FUNCTION_BLOCK FB_AllocateRobotNeedlingMove EXTENDS FB_ActionBasic
VAR_INPUT
    xExecute      : BOOL;
    xAbort        : BOOL;
    TimeOut  : LREAL := 30; // Unit : s
	MovingInfo	: ST_AllocateRobotNeedlingMoveInfo;
END_VAR
VAR_OUTPUT
    xAborted : BOOL;
    iErrorID : INT;
    ErrorMsg : T_MaxString;
END_VAR
VAR
    StateBehavior   : CBML.ETrigATo;
    uiCyclicStep    : UINT := 0;
    uiIndexLoop     : UINT;
	Coordinate		:st_Coordinate;
	fbExecuteEdgeDetect :FB_EdgeDetect;
END_VAR

THIS^.IBehaviourModel := StateBehavior;
StateBehavior(xExecute := xExecute,
              xAbort := xAbort OR fbExecuteEdgeDetect.xFallingEdge,
              udiTimeOut := LREAL_TO_UDINT( TimeOut*1000000),
              xDone => xDone,
              xBusy => xBusy,
              xError => xError,			  
              xAborted => xAborted);			  

			  
//Make sure that C# turns off execute to shut down the service
fbExecuteEdgeDetect(xInput :=xExecute);

//Error Msg
iErrorID := StateBehavior._model.iErrorID;
ErrorMsg := M_GetErrorMsg(xErrorID := iErrorID);

METHOD CleanupAction
VAR_INPUT
    xAbortProposed : BOOL;
    iErrorIDProposed: INT;
END_VAR
VAR_OUTPUT
    xComplete : BOOL := TRUE;
    xAbort: BOOL := xAbortProposed;
 	iErrorID : INT := iErrorIDProposed;
END_VAR
uiCyclicStep := 0;
END_METHOD

METHOD CyclicAction
VAR_INPUT
    itfTimingController : CBML.ITimingController;
END_VAR
VAR_OUTPUT
    xComplete : BOOL := TRUE;
    iErrorID : INT := 0;
END_VAR
VAR_INST
	
END_VAR

VAR
		bAxesCheck 		: BOOL;
	
	
END_VAR
xComplete := FALSE;

	IF arAxisCtrl_gb[AxisNo.Allocate_X].Admin.Axis.Status.Error OR
		arAxisCtrl_gb[AxisNo.Allocate_Y].Admin.Axis.Status.Error THEN
		iErrorID :=3;
	END_IF

CASE uiCyclicStep OF
    0:
		
			uiCyclicStep:=100;
		
		
	100:
			arAxisCtrl_gb[AxisNo.Allocate_X].PosMode.Position:=Coordinate.X;
			arAxisCtrl_gb[AxisNo.Allocate_Y].PosMode.Position:=Coordinate.Y;	
		
			IF arAxisCtrl_gb[AxisNo.Allocate_X].Admin.Axis.Status.Moving OR
			   arAxisCtrl_gb[AxisNo.Allocate_Y].Admin.Axis.Status.Moving OR
			   arAxisStatus_gb[AxisNo.Allocate_X].Admin._OpModeAck=E_AXIS_MODE.ModePosAbs OR
			   arAxisStatus_gb[AxisNo.Allocate_y].Admin._OpModeAck=E_AXIS_MODE.ModePosAbs THEN
			   uiCyclicStep:=200;
			END_IF
			
	200:
			bAxesCheck := TRUE;

		bAxesCheck := bAxesCheck AND	 arAxisStatus_gb[AxisNo.Allocate_x].Admin.CmdDone ;
		bAxesCheck := bAxesCheck AND	 arAxisStatus_gb[AxisNo.Allocate_y].Admin.CmdDone ;	
	
		IF bAxesCheck THEN
			 uiCyclicStep:=600;
		END_IF
	600:
		
		xComplete := TRUE;
END_CASE
END_METHOD

METHOD ExitAction
VAR_INPUT
    xAfterCleanup : BOOL;
    xInCopyCode : BOOL;
END_VAR
END_METHOD

METHOD PRIVATE M_CheckCommand : BOOL
VAR_INPUT
END_VAR
VAR_OUTPUT
	iErrorID	 : INT :=0 ;
END_VAR
VAR
	
END_VAR
IF MovingInfo.Box<0 OR MovingInfo.Box >1 OR MovingInfo.Clip<0 OR MovingInfo.Clip>3 OR MovingInfo.NeedleLocation<0 OR MovingInfo.NeedleLocation>49 THEN
	iErrorID :=2;
	M_CheckCommand := FALSE;
	RETURN;
END_IF

IF MovingInfo.Area = 'T' THEN
		
	FUN_GetNeedleCoordinates(uiLocation :=1 ,
							 uiBox:=MovingInfo.Box,
							 uiClip:=MovingInfo.Clip,
							 uiNeedleLocation:=MovingInfo.NeedleLocation,
							 NeedleCoordinate=>Coordinate);
	IF MovingInfo.Box = 1 AND (MovingInfo.Clip = 2 OR MovingInfo.Clip = 3) THEN
		M_CheckCommand := FALSE;
		iErrorID :=2;
		RETURN;
	END_IF
	IF MovingInfo.Box = 2 AND (MovingInfo.Clip = 0 OR MovingInfo.Clip = 1) THEN
		M_CheckCommand :=FALSE;
		iErrorID :=2;
		RETURN;
	END_IF
	
ELSIF 	

	MovingInfo.Area = 'Q' THEN
	FUN_GetNeedleCoordinates(uiLocation :=0 ,
							 uiBox:=MovingInfo.Box,
							 uiClip:=MovingInfo.Clip,
							 uiNeedleLocation:=MovingInfo.NeedleLocation,
							 NeedleCoordinate=>Coordinate);
	

ELSE
	iErrorID :=2;
	M_CheckCommand := FALSE;
	RETURN;
END_IF

M_CheckCommand:=TRUE;
END_METHOD

METHOD M_GetErrorMsg : T_MaxString
VAR_INPUT
	xErrorID: INT;
END_VAR

VAR
	
END_VAR
CASE xErrorID OF
	0:
		M_GetErrorMsg := 'No Error';
	1:
		M_GetErrorMsg := 'Action time out';
	2:
		M_GetErrorMsg := 'Wrong command';
	3:
		M_GetErrorMsg := 'Servo axis error';
//	4:
//		M_GetErrorMsg := 'Axis roundbelt not ready has Error';
//	5:
//		M_GetErrorMsg := 'Cylinder not ready has Error';
//	6:
//		M_GetErrorMsg := 'Axis RoundBelt has Error';
//	7:
//		M_GetErrorMsg := 'ChargeZone_Plug has Error';
//	8:
//		M_GetErrorMsg := 'TransmitCVZone_Plug has Error';
//	9:
//		M_GetErrorMsg := 'WorkZone_Plug has Error';
//	10:
//		M_GetErrorMsg := 'WorkZone_Press has Error';
END_CASE
END_METHOD

METHOD PRIVATE M_ResetAxes : BOOL
VAR_INPUT
END_VAR
VAR
	bAxesCheck :BOOL;
END_VAR
		bAxesCheck :=TRUE;
		IF arAxisCtrl_gb[AxisNo.Allocate_X].Admin.Axis.Status.Error THEN
			arAxisCtrl_gb[AxisNo.Allocate_X].Admin.ClearError:=TRUE;			
			ELSE
			arAxisCtrl_gb[AxisNo.Allocate_X].Admin.ClearError:=FALSE;	
		END_IF
		IF arAxisCtrl_gb[AxisNo.Allocate_Y].Admin.Axis.Status.Error THEN
			arAxisCtrl_gb[AxisNo.Allocate_Y].Admin.ClearError:=TRUE;			
			ELSE
			arAxisCtrl_gb[AxisNo.Allocate_Y].Admin.ClearError:=FALSE;	
		END_IF
		bAxesCheck := bAxesCheck AND NOT arAxisCtrl_gb[AxisNo.Allocate_X].Admin.ClearError ;
		bAxesCheck := bAxesCheck AND NOT arAxisCtrl_gb[AxisNo.Allocate_X].Admin.ClearError ;
		
		M_ResetAxes := bAxesCheck;
END_METHOD

METHOD ResetAction
VAR_OUTPUT
    xComplete : BOOL := TRUE;
END_VAR
uiCyclicStep := 0;
END_METHOD

METHOD StartAction
VAR_OUTPUT
    xComplete : BOOL := TRUE;
	iErrorID : INT := 0;
END_VAR
xComplete := FALSE;
uiCyclicStep := 0;

IF M_CheckCommand(iErrorID=>iErrorID) AND M_ResetAxes() THEN
	xComplete := TRUE;
END_IF
END_METHOD

END_FUNCTION_BLOCK

(* stored: Version 1.1.0.1, ProductVersion 3.1.4024.13
   POU FB_AllocateRobotNeedlingMove: Id {0c7498d5-c1e2-4999-ae98-a13a68d3d614}, SpecialFunc None
   Folder Action: Id {f2abfd59-5f6d-4076-bcd0-a7a82c0dd92f}
   Method CleanupAction: Id {00a7a5af-0e2b-42d9-87c4-12eebb3a4f46}
   Method CyclicAction: Id {370ca2a2-ffe2-4b71-b033-d8c6b7c21783}
   Method ExitAction: Id {9bf73a84-c586-4ead-be57-22e43bb0f5e5}
   Method M_CheckCommand: Id {8be02945-2678-4ca2-b5e7-c2e375ba11b4}
   Method M_GetErrorMsg: Id {7be2b996-2077-43c1-a6ff-9f7683e73c66}
   Method M_ResetAxes: Id {fefae755-86fa-4863-b4ab-f1ab888f4d16}
   Method ResetAction: Id {90f4d3fa-84d9-441d-858a-cbb8670d3c01}
   Method StartAction: Id {2655a673-413f-4160-b67d-8a355b574926} *)
